// TIA Portal project "Projet3rob" (V15)

(* hardware
DEVICE "Station S7-1200_1"  S7-1200 Station
   slot 0: "Châssis_0"  S7-1200 Rack  Rack  V1.0
   slot 1: "PLC_1"  CPU 1212C DC/DC/DC  6ES7 212-1AE40-0XB0  V4.2
   slot 2: "DI 16/DQ 16x24VDC_1"  6ES7 223-1BL32-0XB0  V2.0
DEVICE "PC-System_1"  SIMATIC PC station
   slot 0: "Station PC SIMATIC"  Rail  SIMATIC PC-Station  V1.0
      slot 125: "Stationmanager"  Station_Manager  V6.0.4
   slot 1: "HMI_RT_1"  WinCC RT Advanced  6AV2 104-0xxxx-xxxx  15.0.0.0
      slot 33792: "Interface hôte"  Host interface
   slot 2: "IE Général_1"  IE General  IE_CP  V8.2.0
*)

// ===== PLC "PLC_1"  CPU 1212C DC/DC/DC =====

VAR_GLOBAL   // PLC tag table "Table de variables standard"
   "System_Byte" AT %MB1 : Byte;
   "FirstScan" AT %M1.0 : Bool;
   "DiagStatusUpdate" AT %M1.1 : Bool;
   "AlwaysTRUE" AT %M1.2 : Bool;
   "AlwaysFALSE" AT %M1.3 : Bool;
   "Clock_Byte" AT %MB0 : Byte;
   "Clock_10Hz" AT %M0.0 : Bool;
   "Clock_5Hz" AT %M0.1 : Bool;
   "Clock_2.5Hz" AT %M0.2 : Bool;
   "Clock_2Hz" AT %M0.3 : Bool;
   "Clock_1.25Hz" AT %M0.4 : Bool;
   "Clock_1Hz" AT %M0.5 : Bool;
   "Clock_0.625Hz" AT %M0.6 : Bool;
   "Clock_0.5Hz" AT %M0.7 : Bool;
   "Q_AUTO_ROBOT_DO_KEP" AT %M22.0 : Bool;
   "ACT_PRODUCT_DO" AT %MW210 : Word;
   "I_ROBOT_DO_KEP" AT %I3.0 : Bool;
   "M_ROBOT_DO_KEP" AT %M13.2 : Bool;
   "Q_MUNU_ROB_DO_KEP" AT %M22.2 : Bool;
END_VAR

VAR_GLOBAL   // PLC tag table "Input"
   "I_Mode" AT %I0.0 : Bool;
   "I_Run" AT %I0.1 : Bool;
   "I_Stop" AT %I0.2 : Bool;
   "I_CB_Vao" AT %I0.3 : Bool;
   "I_CB_Do" AT %I0.4 : Bool;
   "I_CB_Xanh" AT %I0.5 : Bool;
   "I_CB_Do1" AT %I0.6 : Bool;
   "I_CB_Xanh2" AT %I0.7 : Bool;
   "I_CB_Robot_Do_Phai" AT %I1.0 : Bool;
   "I_CB_Robot_Do_Trai" AT %I1.1 : Bool;
   "I_CB_Robot_Do_Giua" AT %I1.2 : Bool;
   "I_CB_Robot_Xanh_Phai" AT %I1.3 : Bool;
   "I_CB_Robot_Xanh_Trai" AT %I1.4 : Bool;
   "I_CB_Robot_Xanh_Giua" AT %I1.5 : Bool;
   "I_BT1" AT %I1.6 : Bool;
   "I_BT2" AT %I1.7 : Bool;
   "I_Xylanh_Do" AT %I2.0 : Bool;
   "I_Xylanh_Xanh" AT %I2.1 : Bool;
   "I_Robot_Do_Trai" AT %I2.2 : Bool;
   "I_Robot_Do_Phai" AT %I2.3 : Bool;
   "I_Robot_Do_Glua" AT %I2.4 : Bool;
   "I_Robot_Xanh_Trai" AT %I2.5 : Bool;
   "I_Robot_Xanh_Phai" AT %I2.6 : Bool;
   "I_Robot_Xanh_Glua" AT %I2.7 : Bool;
END_VAR

VAR_GLOBAL   // PLC tag table "M"
   "M_Mode" AT %M10.0 : Bool;
   "M_Run" AT %M10.1 : Bool;
   "M_Stop" AT %M10.2 : Bool;
   "M_CB_Vao" AT %M10.3 : Bool;
   "M_CB_Do" AT %M10.4 : Bool;
   "M_CB_Xanh" AT %M10.5 : Bool;
   "M_CB_Do1" AT %M10.6 : Bool;
   "M_CB_Xanh2" AT %M10.7 : Bool;
   "M_CB_Robot_Do_Phai" AT %M11.0 : Bool;
   "M_CB_Robot_Do_Trai" AT %M11.1 : Bool;
   "M_CB_Robot_Do_Giua" AT %M11.2 : Bool;
   "M_CB_Robot_Xanh_Phai" AT %M11.3 : Bool;
   "M_CB_Robot_Xanh_Trai" AT %M11.4 : Bool;
   "M_CB_Robot_Xanh_Giua" AT %M11.5 : Bool;
   "M_BT1" AT %M11.6 : Bool;
   "M_BT2" AT %M11.7 : Bool;
   "M_Xylanh_Do" AT %M12.0 : Bool;
   "M_Xylanh_Xanh" AT %M12.1 : Bool;
   "M_Robot_Do_Trai" AT %M12.2 : Bool;
   "M_Robot_Do_Phai" AT %M12.3 : Bool;
   "M_Robot_Do_Glua" AT %M12.4 : Bool;
   "M_Robot_Xanh_Trai" AT %M12.5 : Bool;
   "M_Robot_Xanh_Phai" AT %M12.6 : Bool;
   "M_Robot_Xanh_Glua" AT %M12.7 : Bool;
   "M_Simulation" AT %M13.0 : Bool;
   "M_Reset" AT %M13.1 : Bool;
END_VAR

VAR_GLOBAL   // PLC tag table "OUTPUT"
   "Q_Lamp_Auto" AT %Q0.0 : Bool;
   "Q_Lamp_Manu" AT %Q0.1 : Bool;
   "Q_Lamp_Running" AT %Q0.2 : Bool;
   "Q_Lamp_Stop" AT %Q0.3 : Bool;
   "Q_BT1" AT %Q0.4 : Bool;
   "Q_BT2" AT %Q0.5 : Bool;
   "Q_Xylanh_Do" AT %Q0.6 : Bool;
   "Q_Xylanh_Xanh" AT %Q0.7 : Bool;
   "Q_Robot_Do_Trai" AT %Q1.0 : Bool;
   "Q_Robot_Do_Phai" AT %Q1.1 : Bool;
   "Q_Robot_Xanh_Trai" AT %Q1.2 : Bool;
   "Q_Robot_Xanh_Phai" AT %Q1.3 : Bool;
END_VAR

VAR_GLOBAL   // PLC tag table "Xlanh P"
   "P1" AT %M40.0 : Bool;
   "P2" AT %M40.1 : Bool;
   "P3" AT %M40.2 : Bool;
   "P4" AT %M40.3 : Bool;
   "P5" AT %M40.4 : Bool;
   "P6" AT %M40.5 : Bool;
   "P7" AT %M40.6 : Bool;
   "P8" AT %M40.7 : Bool;
   "P9" AT %M41.0 : Bool;
   "P10" AT %M41.1 : Bool;
   "P11" AT %M41.2 : Bool;
   "P12" AT %M41.3 : Bool;
   "P13" AT %M41.4 : Bool;
   "P14" AT %M41.5 : Bool;
   "P15" AT %M41.6 : Bool;
   "P16" AT %M41.7 : Bool;
   "P17" AT %M42.0 : Bool;
   "P18" AT %M42.1 : Bool;
   "P19" AT %M42.2 : Bool;
   "P20" AT %M42.3 : Bool;
   "P21" AT %M42.4 : Bool;
   "P22" AT %M42.5 : Bool;
   "P23" AT %M42.6 : Bool;
   "P24" AT %M42.7 : Bool;
   "P25" AT %M43.0 : Bool;
   "P26" AT %M43.1 : Bool;
   "P27" AT %M43.2 : Bool;
   "P28" AT %M43.3 : Bool;
   "P29" AT %M43.4 : Bool;
   "P30" AT %M43.5 : Bool;
END_VAR

VAR_GLOBAL   // PLC tag table "TRING GIAN"
   "Q_Auto_BT1" AT %M20.0 : Bool;
   "Q_Auto_BT2" AT %M20.1 : Bool;
   "Q_Auto_Xylanh_Do" AT %M20.2 : Bool;
   "Q_Auto_Xylanh_Xanh" AT %M20.3 : Bool;
   "Q_Auto_Robot_Do_Trai" AT %M20.4 : Bool;
   "Q_Auto_Robot_Do_Phai" AT %M20.5 : Bool;
   "Q_Auto_Robot_Xanh_Trai" AT %M20.6 : Bool;
   "Q_Auto_Robot_Xanh_Phai" AT %M20.7 : Bool;
   "Q_Manu_BT1" AT %M21.0 : Bool;
   "Q_Manu_BT2" AT %M21.1 : Bool;
   "Q_Manu_Xylanh_Do" AT %M21.2 : Bool;
   "Q_Manu_Xylanh_Xanh" AT %M21.3 : Bool;
   "Q_Manu_Robot_Do_Trai" AT %M21.4 : Bool;
   "Q_Manu_Robot_Do_Phai" AT %M21.5 : Bool;
   "Q_Manu_Robot_Xanh_Trai" AT %M21.6 : Bool;
   "Q_Manu_Robot_Xanh_Phai" AT %M21.7 : Bool;
END_VAR

VAR_GLOBAL   // PLC tag table "DU MUE"
   "Act_Count_Vao" AT %MW200 : Int;
   "Act_Count_Do" AT %MW202 : Int;
   "Act_Count_Do1" AT %MW204 : Int;
   "Act_Count_Xnah" AT %MW206 : Int;
   "Act_Count_Xnah1" AT %MW208 : Int;
END_VAR

VAR_GLOBAL   // PLC tag table "Table de variables_1"
   "ROBOT_DO_AUTO_STEP1" AT %M25.0 : Bool;
   "ROBOT_DO_AUTO_STEP2" AT %M25.1 : Bool;
   "ROBOT_DO_AUTO_STEP3" AT %M25.2 : Bool;
   "ROBOT_DO_AUTO_STEP4" AT %M25.3 : Bool;
   "ROBOT_DO_AUTO_STEP5" AT %M25.4 : Bool;
   "ROBOT_XNAH_AUTO_STEP1" AT %M25.5 : Bool;
   "ROBOT_XNAH_AUTO_STEP2" AT %M25.6 : Bool;
   "ROBOT_XNAH_AUTO_STEP3" AT %M25.7 : Bool;
   "ROBOT_XNAH_AUTO_STEP4" AT %M26.0 : Bool;
   "ROBOT_XNAH_AUTO_STEP5" AT %M26.1 : Bool;
END_VAR

// folder: System blocks/Program resources

DATA_BLOCK "IEC_Timer_0_DB"   // DB1
{ S7_Optimized_Access := 'TRUE' }
AUTHOR : Simatic
FAMILY : IEC
NAME : IEC_TMR
VERSION : 1.0
// stored: InstanceOfName IEC_TIMER
"IEC_TIMER"
BEGIN
END_DATA_BLOCK

DATA_BLOCK "TIMER_DELYE_SET_XL_DO"   // DB2
{ S7_Optimized_Access := 'TRUE' }
AUTHOR : Simatic
FAMILY : IEC
NAME : IEC_TMR
VERSION : 1.0
// stored: InstanceOfName IEC_TIMER
"IEC_TIMER"
BEGIN
END_DATA_BLOCK

DATA_BLOCK "TIMER_XL_DO"   // DB3
{ S7_Optimized_Access := 'TRUE' }
AUTHOR : Simatic
FAMILY : IEC
NAME : IEC_TMR
VERSION : 1.0
// stored: InstanceOfName IEC_TIMER
"IEC_TIMER"
BEGIN
END_DATA_BLOCK

DATA_BLOCK "TIME_KEP_DO1"   // DB4
{ S7_Optimized_Access := 'TRUE' }
AUTHOR : Simatic
FAMILY : IEC
NAME : IEC_TMR
VERSION : 1.0
// stored: InstanceOfName IEC_TIMER
"IEC_TIMER"
BEGIN
END_DATA_BLOCK

DATA_BLOCK "TIMER_KEP_DO2"   // DB5
{ S7_Optimized_Access := 'TRUE' }
AUTHOR : Simatic
FAMILY : IEC
NAME : IEC_TMR
VERSION : 1.0
// stored: InstanceOfName IEC_TIMER
"IEC_TIMER"
BEGIN
END_DATA_BLOCK

DATA_BLOCK "IEC_Timer_0_DB_1"   // DB6
{ S7_Optimized_Access := 'TRUE' }
AUTHOR : Simatic
FAMILY : IEC
NAME : IEC_TMR
VERSION : 1.0
// stored: InstanceOfName IEC_TIMER
"IEC_TIMER"
BEGIN
END_DATA_BLOCK

DATA_BLOCK "TIMER_DELYE_SET_XL_XNAH"   // DB7
{ S7_Optimized_Access := 'TRUE' }
AUTHOR : Simatic
FAMILY : IEC
NAME : IEC_TMR
VERSION : 1.0
// stored: InstanceOfName IEC_TIMER
"IEC_TIMER"
BEGIN
END_DATA_BLOCK

DATA_BLOCK "TIMER_XL_XANH"   // DB8
{ S7_Optimized_Access := 'TRUE' }
AUTHOR : Simatic
FAMILY : IEC
NAME : IEC_TMR
VERSION : 1.0
// stored: InstanceOfName IEC_TIMER
"IEC_TIMER"
BEGIN
END_DATA_BLOCK

// folder: (top level)

FUNCTION "FC_Auto" : Void   // FC1, LAD
{ S7_Optimized_Access := 'TRUE' }
VERSION : 0.1
   VAR_TEMP   // added for the SCL form of the ladder/FBD networks
      _w1 : Bool;
      _w2 : Bool;
      _w3 : Bool;
      _w4 : Bool;
      _w5 : Bool;
      _w6 : Bool;
      _w7 : Bool;
      _w8 : Bool;
      _w9 : Bool;
      _w10 : Bool;
      _w11 : Bool;
      _w12 : Bool;
      _w13 : Bool;
      _w14 : Bool;
   END_VAR
BEGIN

REGION Network 1
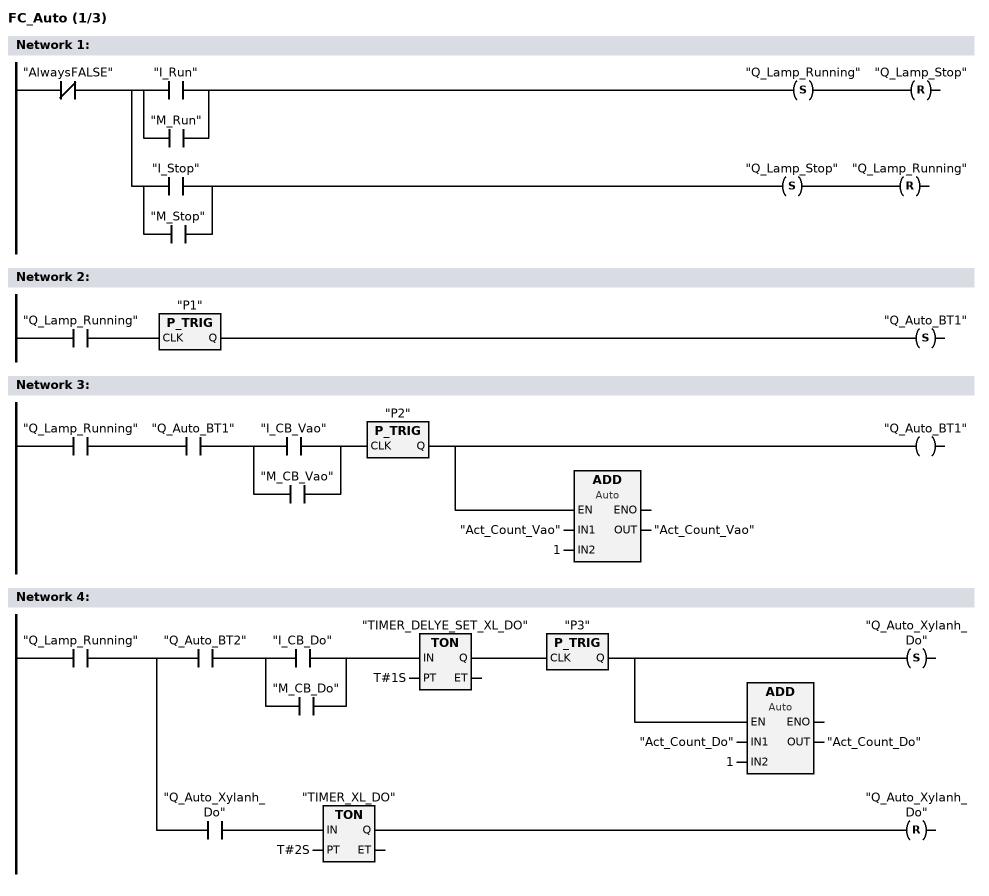
   RUNG wire#powerrail
      I_Contact( "AlwaysFALSE" )
      wire#w1
      Contact( "I_Run" )
      wire#w2
      S_Coil( "Q_Lamp_Running" )
      R_Coil( "Q_Lamp_Stop" )
   END_RUNG
   RUNG wire#w1
      Contact( "M_Run" )
   END_RUNG wire#w2
   RUNG wire#w1
      Contact( "I_Stop" )
      wire#w3
      S_Coil( "Q_Lamp_Stop" )
      R_Coil( "Q_Lamp_Running" )
   END_RUNG
   RUNG wire#w1
      Contact( "M_Stop" )
   END_RUNG wire#w3
   // the same network as SCL:
   IF NOT "AlwaysFALSE" AND ("I_Run" OR "M_Run") THEN
       "Q_Lamp_Running" := TRUE;
       "Q_Lamp_Stop" := FALSE;
   END_IF;
   IF NOT "AlwaysFALSE" AND ("I_Stop" OR "M_Stop") THEN
       "Q_Lamp_Stop" := TRUE;
       "Q_Lamp_Running" := FALSE;
   END_IF;
END_REGION

REGION Network 2
   RUNG wire#powerrail
      Contact( "Q_Lamp_Running" )
      P_Trig( "P1" )
      S_Coil( "Q_Auto_BT1" )
   END_RUNG
   // the same network as SCL:
   #_w1 := "Q_Lamp_Running" AND NOT "P1";   // rising edge
   "P1" := "Q_Lamp_Running";
   IF #_w1 THEN "Q_Auto_BT1" := TRUE; END_IF;
END_REGION

REGION Network 3
   RUNG wire#powerrail
      Contact( "Q_Lamp_Running" )
      Contact( "Q_Auto_BT1" )
      wire#w1
      Contact( "I_CB_Vao" )
      wire#w2
      P_Trig( "P2" )
      wire#w3
      Coil( "Q_Auto_BT1" )
   END_RUNG
   RUNG wire#w1
      Contact( "M_CB_Vao" )
   END_RUNG wire#w2
   RUNG wire#w3
      Add(in1 := "Act_Count_Vao", in2 := 1, out => "Act_Count_Vao")
   END_RUNG
   // the same network as SCL:
   #_w1 := "Q_Lamp_Running" AND "Q_Auto_BT1" AND ("I_CB_Vao" OR "M_CB_Vao");
   #_w2 := #_w1 AND NOT "P2";   // rising edge
   "P2" := #_w1;
   "Q_Auto_BT1" := #_w2;
   IF #_w2 THEN "Act_Count_Vao" := "Act_Count_Vao" + 1; END_IF;
END_REGION

REGION Network 4
   "TIMER_DELYE_SET_XL_DO".TON(IN := "Q_Lamp_Running" AND "Q_Auto_BT2" AND ("I_CB_Do" OR "M_CB_Do"), PT := T#1S);
   #_w1 := "TIMER_DELYE_SET_XL_DO".Q AND NOT "P3";   // rising edge
   "P3" := "TIMER_DELYE_SET_XL_DO".Q;
   IF #_w1 THEN
       "Q_Auto_Xylanh_Do" := TRUE;
       "Act_Count_Do" := "Act_Count_Do" + 1;
   END_IF;
   "TIMER_XL_DO".TON(IN := "Q_Lamp_Running" AND "Q_Auto_Xylanh_Do", PT := T#2S);
   IF "TIMER_XL_DO".Q THEN "Q_Auto_Xylanh_Do" := FALSE; END_IF;
END_REGION

REGION Network 5
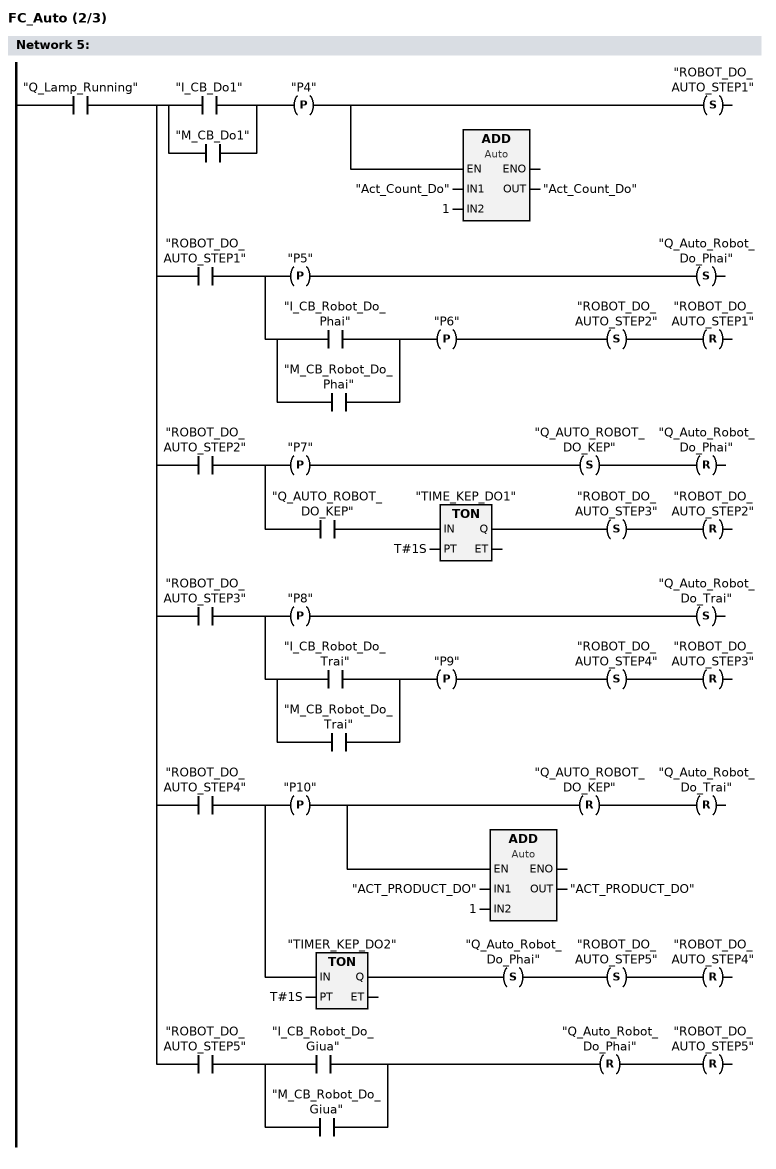
   #_w1 := "Q_Lamp_Running" AND ("I_CB_Do1" OR "M_CB_Do1");
   #_w2 := #_w1 AND NOT "P4";   // rising edge
   "P4" := #_w1;
   IF #_w2 THEN
       "ROBOT_DO_AUTO_STEP1" := TRUE;
       "Act_Count_Do" := "Act_Count_Do" + 1;
   END_IF;
   #_w3 := "Q_Lamp_Running" AND "ROBOT_DO_AUTO_STEP1";
   #_w4 := #_w3 AND NOT "P5";   // rising edge
   "P5" := #_w3;
   IF #_w4 THEN "Q_Auto_Robot_Do_Phai" := TRUE; END_IF;
   #_w5 := #_w3 AND ("I_CB_Robot_Do_Phai" OR "M_CB_Robot_Do_Phai");
   #_w6 := #_w5 AND NOT "P6";   // rising edge
   "P6" := #_w5;
   IF #_w6 THEN
       "ROBOT_DO_AUTO_STEP2" := TRUE;
       "ROBOT_DO_AUTO_STEP1" := FALSE;
   END_IF;
   #_w7 := "Q_Lamp_Running" AND "ROBOT_DO_AUTO_STEP2";
   #_w8 := #_w7 AND NOT "P7";   // rising edge
   "P7" := #_w7;
   IF #_w8 THEN
       "Q_AUTO_ROBOT_DO_KEP" := TRUE;
       "Q_Auto_Robot_Do_Phai" := FALSE;
   END_IF;
   "TIME_KEP_DO1".TON(IN := #_w7 AND "Q_AUTO_ROBOT_DO_KEP", PT := T#1S);
   IF "TIME_KEP_DO1".Q THEN
       "ROBOT_DO_AUTO_STEP3" := TRUE;
       "ROBOT_DO_AUTO_STEP2" := FALSE;
   END_IF;
   #_w9 := "Q_Lamp_Running" AND "ROBOT_DO_AUTO_STEP3";
   #_w10 := #_w9 AND NOT "P8";   // rising edge
   "P8" := #_w9;
   IF #_w10 THEN "Q_Auto_Robot_Do_Trai" := TRUE; END_IF;
   #_w11 := #_w9 AND ("I_CB_Robot_Do_Trai" OR "M_CB_Robot_Do_Trai");
   #_w12 := #_w11 AND NOT "P9";   // rising edge
   "P9" := #_w11;
   IF #_w12 THEN
       "ROBOT_DO_AUTO_STEP4" := TRUE;
       "ROBOT_DO_AUTO_STEP3" := FALSE;
   END_IF;
   #_w13 := "Q_Lamp_Running" AND "ROBOT_DO_AUTO_STEP4";
   #_w14 := #_w13 AND NOT "P10";   // rising edge
   "P10" := #_w13;
   IF #_w14 THEN
       "Q_AUTO_ROBOT_DO_KEP" := FALSE;
       "Q_Auto_Robot_Do_Trai" := FALSE;
       "ACT_PRODUCT_DO" := "ACT_PRODUCT_DO" + 1;
   END_IF;
   "TIMER_KEP_DO2".TON(IN := #_w13, PT := T#1S);
   IF "TIMER_KEP_DO2".Q THEN
       "Q_Auto_Robot_Do_Phai" := TRUE;
       "ROBOT_DO_AUTO_STEP5" := TRUE;
       "ROBOT_DO_AUTO_STEP4" := FALSE;
   END_IF;
   IF "Q_Lamp_Running" AND "ROBOT_DO_AUTO_STEP5" AND ("I_CB_Robot_Do_Giua" OR "M_CB_Robot_Do_Giua") THEN
       "Q_Auto_Robot_Do_Phai" := FALSE;
       "ROBOT_DO_AUTO_STEP5" := FALSE;
   END_IF;
END_REGION

REGION Network 6
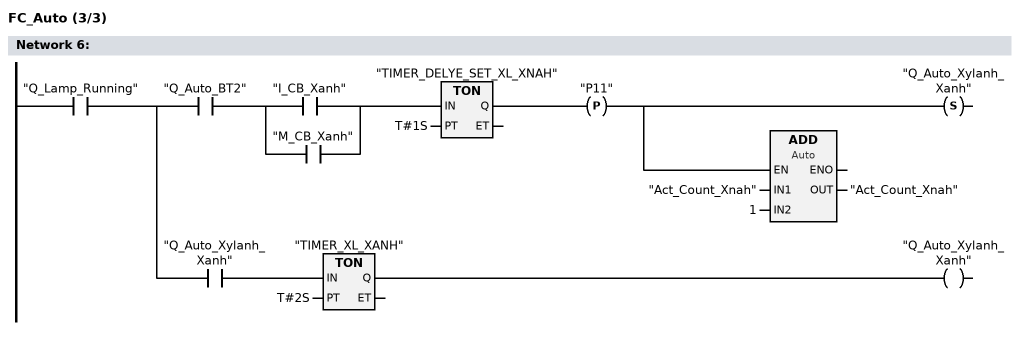
   "TIMER_DELYE_SET_XL_XNAH".TON(IN := "Q_Lamp_Running" AND "Q_Auto_BT2" AND ("I_CB_Xanh" OR "M_CB_Xanh"),
                           PT := T#1S);
   #_w1 := "TIMER_DELYE_SET_XL_XNAH".Q AND NOT "P11";   // rising edge
   "P11" := "TIMER_DELYE_SET_XL_XNAH".Q;
   IF #_w1 THEN
       "Q_Auto_Xylanh_Xanh" := TRUE;
       "Act_Count_Xnah" := "Act_Count_Xnah" + 1;
   END_IF;
   "TIMER_XL_XANH".TON(IN := "Q_Lamp_Running" AND "Q_Auto_Xylanh_Xanh", PT := T#2S);
   "Q_Auto_Xylanh_Xanh" := "TIMER_XL_XANH".Q;
END_REGION
END_FUNCTION

FUNCTION "FC_Manu" : Void   // FC2, LAD
{ S7_Optimized_Access := 'TRUE' }
VERSION : 0.1
   VAR_TEMP   // added for the SCL form of the ladder/FBD networks
      _w1 : Bool;
      _w2 : Bool;
      _w3 : Bool;
      _w4 : Bool;
   END_VAR
BEGIN

REGION Network 1
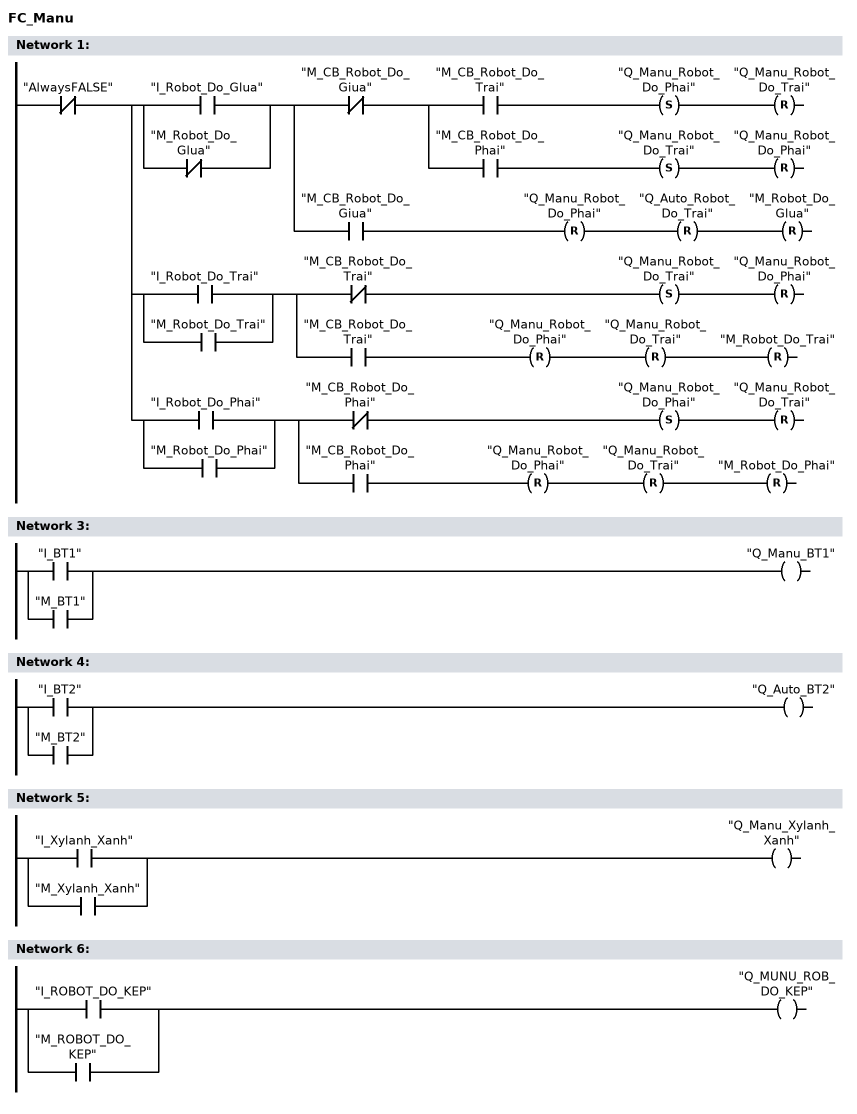
   RUNG wire#powerrail
      I_Contact( "AlwaysFALSE" )
      wire#w1
      Contact( "I_Robot_Do_Glua" )
      wire#w2
      I_Contact( "M_CB_Robot_Do_Giua" )
      wire#w3
      Contact( "M_CB_Robot_Do_Trai" )
      S_Coil( "Q_Manu_Robot_Do_Phai" )
      R_Coil( "Q_Manu_Robot_Do_Trai" )
   END_RUNG
   RUNG wire#w1
      I_Contact( "M_Robot_Do_Glua" )
   END_RUNG wire#w2
   RUNG wire#w3
      Contact( "M_CB_Robot_Do_Phai" )
      S_Coil( "Q_Manu_Robot_Do_Trai" )
      R_Coil( "Q_Manu_Robot_Do_Phai" )
   END_RUNG
   RUNG wire#w2
      Contact( "M_CB_Robot_Do_Giua" )
      R_Coil( "Q_Manu_Robot_Do_Phai" )
      R_Coil( "Q_Auto_Robot_Do_Trai" )
      R_Coil( "M_Robot_Do_Glua" )
   END_RUNG
   RUNG wire#w1
      Contact( "I_Robot_Do_Trai" )
      wire#w4
      I_Contact( "M_CB_Robot_Do_Trai" )
      S_Coil( "Q_Manu_Robot_Do_Trai" )
      R_Coil( "Q_Manu_Robot_Do_Phai" )
   END_RUNG
   RUNG wire#w1
      Contact( "M_Robot_Do_Trai" )
   END_RUNG wire#w4
   RUNG wire#w4
      Contact( "M_CB_Robot_Do_Trai" )
      R_Coil( "Q_Manu_Robot_Do_Phai" )
      R_Coil( "Q_Manu_Robot_Do_Trai" )
      R_Coil( "M_Robot_Do_Trai" )
   END_RUNG
   RUNG wire#w1
      Contact( "I_Robot_Do_Phai" )
      wire#w5
      I_Contact( "M_CB_Robot_Do_Phai" )
      S_Coil( "Q_Manu_Robot_Do_Phai" )
      R_Coil( "Q_Manu_Robot_Do_Trai" )
   END_RUNG
   RUNG wire#w1
      Contact( "M_Robot_Do_Phai" )
   END_RUNG wire#w5
   RUNG wire#w5
      Contact( "M_CB_Robot_Do_Phai" )
      R_Coil( "Q_Manu_Robot_Do_Phai" )
      R_Coil( "Q_Manu_Robot_Do_Trai" )
      R_Coil( "M_Robot_Do_Phai" )
   END_RUNG
   // the same network as SCL:
   #_w1 := NOT "AlwaysFALSE" AND ("I_Robot_Do_Glua" OR NOT "M_Robot_Do_Glua");
   #_w2 := #_w1 AND NOT "M_CB_Robot_Do_Giua";
   IF #_w2 AND "M_CB_Robot_Do_Trai" THEN
       "Q_Manu_Robot_Do_Phai" := TRUE;
       "Q_Manu_Robot_Do_Trai" := FALSE;
   END_IF;
   IF #_w2 AND "M_CB_Robot_Do_Phai" THEN
       "Q_Manu_Robot_Do_Trai" := TRUE;
       "Q_Manu_Robot_Do_Phai" := FALSE;
   END_IF;
   IF #_w1 AND "M_CB_Robot_Do_Giua" THEN
       "Q_Manu_Robot_Do_Phai" := FALSE;
       "Q_Auto_Robot_Do_Trai" := FALSE;
       "M_Robot_Do_Glua" := FALSE;
   END_IF;
   #_w3 := NOT "AlwaysFALSE" AND ("I_Robot_Do_Trai" OR "M_Robot_Do_Trai");
   IF #_w3 AND NOT "M_CB_Robot_Do_Trai" THEN
       "Q_Manu_Robot_Do_Trai" := TRUE;
       "Q_Manu_Robot_Do_Phai" := FALSE;
   END_IF;
   IF #_w3 AND "M_CB_Robot_Do_Trai" THEN
       "Q_Manu_Robot_Do_Phai" := FALSE;
       "Q_Manu_Robot_Do_Trai" := FALSE;
       "M_Robot_Do_Trai" := FALSE;
   END_IF;
   #_w4 := NOT "AlwaysFALSE" AND ("I_Robot_Do_Phai" OR "M_Robot_Do_Phai");
   IF #_w4 AND NOT "M_CB_Robot_Do_Phai" THEN
       "Q_Manu_Robot_Do_Phai" := TRUE;
       "Q_Manu_Robot_Do_Trai" := FALSE;
   END_IF;
   IF #_w4 AND "M_CB_Robot_Do_Phai" THEN
       "Q_Manu_Robot_Do_Phai" := FALSE;
       "Q_Manu_Robot_Do_Trai" := FALSE;
       "M_Robot_Do_Phai" := FALSE;
   END_IF;
END_REGION

REGION Network 3
   RUNG wire#powerrail
      Contact( "I_BT1" )
      wire#w1
      Coil( "Q_Manu_BT1" )
   END_RUNG
   RUNG wire#powerrail
      Contact( "M_BT1" )
   END_RUNG wire#w1
   // the same network as SCL:
   "Q_Manu_BT1" := "I_BT1" OR "M_BT1";
END_REGION

REGION Network 4
   RUNG wire#powerrail
      Contact( "I_BT2" )
      wire#w1
      Coil( "Q_Auto_BT2" )
   END_RUNG
   RUNG wire#powerrail
      Contact( "M_BT2" )
   END_RUNG wire#w1
   // the same network as SCL:
   "Q_Auto_BT2" := "I_BT2" OR "M_BT2";
END_REGION

REGION Network 5
   RUNG wire#powerrail
      Contact( "I_Xylanh_Xanh" )
      wire#w1
      Coil( "Q_Manu_Xylanh_Xanh" )
   END_RUNG
   RUNG wire#powerrail
      Contact( "M_Xylanh_Xanh" )
   END_RUNG wire#w1
   // the same network as SCL:
   "Q_Manu_Xylanh_Xanh" := "I_Xylanh_Xanh" OR "M_Xylanh_Xanh";
END_REGION

REGION Network 6
   RUNG wire#powerrail
      Contact( "I_ROBOT_DO_KEP" )
      wire#w1
      Coil( "Q_MUNU_ROB_DO_KEP" )
   END_RUNG
   RUNG wire#powerrail
      Contact( "M_ROBOT_DO_KEP" )
   END_RUNG wire#w1
   // the same network as SCL:
   "Q_MUNU_ROB_DO_KEP" := "I_ROBOT_DO_KEP" OR "M_ROBOT_DO_KEP";
END_REGION
END_FUNCTION

FUNCTION "FC_SIMULATION" : Void   // FC3, LAD
{ S7_Optimized_Access := 'TRUE' }
VERSION : 0.1
BEGIN
END_FUNCTION

FUNCTION "FC_OUTPUT" : Void   // FC4, LAD
{ S7_Optimized_Access := 'TRUE' }
VERSION : 0.1
BEGIN
END_FUNCTION

ORGANIZATION_BLOCK "Main"   // OB1, LAD, ProgramCycle
TITLE = "Main Program Sweep (Cycle)"
{ S7_Optimized_Access := 'TRUE' }
VERSION : 0.1
   VAR_INPUT
      Initial_Call : Bool;   // Initial call of this OB
      Remanence : Bool;   // =True, if remanent data are available
   END_VAR
BEGIN

REGION Network 1
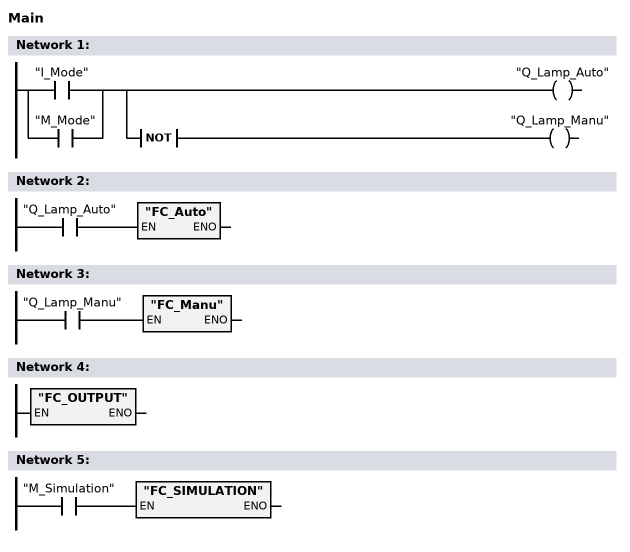
   RUNG wire#powerrail
      Contact( "I_Mode" )
      wire#w1
      Coil( "Q_Lamp_Auto" )
   END_RUNG
   RUNG wire#powerrail
      Contact( "M_Mode" )
   END_RUNG wire#w1
   RUNG wire#w1
      Not()
      Coil( "Q_Lamp_Manu" )
   END_RUNG
   // the same network as SCL:
   "Q_Lamp_Auto" := "I_Mode" OR "M_Mode";
   "Q_Lamp_Manu" := NOT "Q_Lamp_Auto";
END_REGION

REGION Network 2
   RUNG wire#powerrail
      Contact( "Q_Lamp_Auto" )
      "FC_Auto"()
   END_RUNG
   // the same network as SCL:
   IF "Q_Lamp_Auto" THEN "FC_Auto"(); END_IF;
END_REGION

REGION Network 3
   RUNG wire#powerrail
      Contact( "Q_Lamp_Manu" )
      "FC_Manu"()
   END_RUNG
   // the same network as SCL:
   IF "Q_Lamp_Manu" THEN "FC_Manu"(); END_IF;
END_REGION

REGION Network 4
   RUNG wire#powerrail
      "FC_OUTPUT"()
   END_RUNG
   // the same network as SCL:
   "FC_OUTPUT"();
END_REGION

REGION Network 5
   RUNG wire#powerrail
      Contact( "M_Simulation" )
      "FC_SIMULATION"()
   END_RUNG
   // the same network as SCL:
   IF "M_Simulation" THEN "FC_SIMULATION"(); END_IF;
END_REGION
END_ORGANIZATION_BLOCK

ORGANIZATION_BLOCK "Startup"   // OB100, LAD, Startup
TITLE = "Complete Restart"
{ S7_Optimized_Access := 'TRUE' }
VERSION : 0.1
   VAR_INPUT
      LostRetentive : Bool;   // True if retentive data are lost
      LostRTC : Bool;   // True if date and time are lost
   END_VAR
BEGIN
END_ORGANIZATION_BLOCK

(* ===== HMI "HMI_RT_1" =====
system functions are stored by id; their names below are inferred from use
connection "HMI_Liaison_1": ETHERNET, S7_1200_OMS

HMI tags "Table de variables standard"
   "Q_BT2" : Bool = PLC Q_BT2 AT %Q0.5, 1 s
   "Q_BT1" : Bool = PLC Q_BT1 AT %Q0.4, 1 s
   "M_CB_Vao" : Bool = PLC M_CB_Vao AT %M10.3, 1 s
   "M_CB_Do" : Bool = PLC M_CB_Do AT %M10.4, 1 s
   "M_CB_Xanh" : Bool = PLC M_CB_Xanh AT %M10.5, 1 s
   "M_CB_Do1" : Bool = PLC M_CB_Do1 AT %M10.6, 1 s
   "M_CB_Xanh1" : Bool = PLC M_CB_Xanh2 AT %M10.7, 1 s
   "M_CB_Robot_Do_Trai" : Bool = PLC M_CB_Robot_Do_Trai AT %M11.1, 1 s
   "M_CB_Robot_Do_Giua" : Bool = PLC M_CB_Robot_Do_Giua AT %M11.2, 1 s
   "M_CB_Robot_Do_Phai" : Bool = PLC M_CB_Robot_Do_Phai AT %M11.0, 1 s
   "M_CB_Robot_Xanh_Trai" : Bool = PLC M_CB_Robot_Xanh_Trai AT %M11.4, 1 s
   "M_CB_Robot_Xanh_Giua" : Bool = PLC M_CB_Robot_Xanh_Giua AT %M11.5, 1 s
   "M_CB_Robot_Xanh_Phai" : Bool = PLC M_CB_Robot_Xanh_Phai AT %M11.3, 1 s
   "Q_Xylanh_Do" : Bool = PLC Q_Xylanh_Do AT %Q0.6, 1 s
   "Q_Xylanh_Xanh" : Bool = PLC Q_Xylanh_Xanh AT %Q0.7, 1 s
   "M_Simulation" : Bool = PLC M_Simulation AT %M13.0, 1 s
   "M_Mode" : Bool = PLC M_Mode AT %M10.0, 1 s
   "M_Run" : Bool = PLC M_Run AT %M10.1, 1 s
   "M_Stop" : Bool = PLC M_Stop AT %M10.2, 1 s
   "M_Reset" : Bool = PLC M_Reset AT %M13.1, 1 s
   "Q_Lamp_Auto" : Bool = PLC Q_Lamp_Auto AT %Q0.0, 1 s
   "Q_Lamp_Manu" : Bool = PLC Q_Lamp_Manu AT %Q0.1, 1 s
   "Q_Lamp_Running" : Bool = PLC Q_Lamp_Running AT %Q0.2, 1 s
   "Q_Lamp_Stop" : Bool = PLC Q_Lamp_Stop AT %Q0.3, 1 s
   "M_BT1" : Bool = PLC M_BT1 AT %M11.6, 1 s
   "M_BT2" : Bool = PLC M_BT2 AT %M11.7, 1 s
   "M_Xylanh_Do" : Bool = PLC M_Xylanh_Do AT %M12.0, 1 s
   "M_Xylanh_Xanh" : Bool = PLC M_Xylanh_Xanh AT %M12.1, 1 s
   "M_Robot_Do_Phai" : Bool = PLC M_Robot_Do_Phai AT %M12.3, 1 s
   "M_Robot_Do_Glua" : Bool = PLC M_Robot_Do_Glua AT %M12.4, 1 s
   "M_Robot_Do_Trai" : Bool = PLC M_Robot_Do_Trai AT %M12.2, 1 s
   "M_Robot_Xanh_Phai" : Bool = PLC M_Robot_Xanh_Phai AT %M12.6, 1 s
   "M_Robot_Xanh_Glua" : Bool = PLC M_Robot_Xanh_Glua AT %M12.7, 1 s
   "M_Robot_Xanh_Trai" : Bool = PLC M_Robot_Xanh_Trai AT %M12.5, 1 s
   "Q_Robot_Xanh_Trai" : Bool = PLC Q_Robot_Xanh_Trai AT %Q1.2, 1 s
   "Q_Robot_Xanh_Phai" : Bool = PLC Q_Robot_Xanh_Phai AT %Q1.3, 1 s
   "Q_Robot_Do_Trai" : Bool = PLC Q_Robot_Do_Trai AT %Q1.0, 1 s
   "Q_Robot_Do_Phai" : Bool = PLC Q_Robot_Do_Phai AT %Q1.1, 1 s

screen "Vue_1" 1024x1280
   TextField "Champ de texte_1" at 370,18 size 186x22; Text 'TIA PORTAL + S7-1200'
   SymbolLibrary "Bibliothèque des icônes_2" at 257,256 size 212x54
      Appearance <- "Q_BT2"
   SymbolLibrary "Bibliothèque des icônes_3" at 436,255 size 215x54
      Appearance <- "Q_BT2"
   SymbolLibrary "Bibliothèque des icônes_4" at 21,251 size 263x54
      Appearance <- "Q_BT1"
   SymbolLibrary "Bibliothèque des icônes_5" at 172,181 size 27x47
      Appearance <- "M_CB_Vao"
   SymbolLibrary "Bibliothèque des icônes_6" at 37,308 size 57x60
      Appearance <- "Q_BT1"
   SymbolLibrary "Bibliothèque des icônes_8" at 358,176 size 27x57
      Appearance <- "M_CB_Do"
   Group "Group_2" at 434,141 size 78x66
   Polygon "Polygone_7" at 247,376 size 114x77
      Visibility <- "M_CB_Robot_Do_Phai"
   Polygon "Polygone_10" at 125,410 size 124x46
      Visibility <- "M_CB_Robot_Do_Trai"
   Rectangle "Rectangle_9" at 248,409 size 20x45
      Visibility <- "M_CB_Robot_Do_Giua"
   Circle "Cercle_2" at 333,420 size 10x10
      Appearance <- "M_CB_Robot_Do_Phai"
   Circle "Cercle_4" at 251,410 size 10x10
      Appearance <- "M_CB_Robot_Do_Giua"
   Circle "Cercle_5" at 151,428 size 10x10
      Appearance <- "M_CB_Robot_Do_Trai"
   SymbolLibrary "Bibliothèque des icônes_9" at 70,437 size 87x60
   SymbolLibrary "Bibliothèque des icônes_10" at 370,364 size 69x29
      Appearance <- "M_CB_Do1"
   IOField "Champ d'E/S_1" at 37,157 size 96x32; FormatPattern 9999999
   IOField "Champ d'E/S_2" at 330,141 size 96x32; FormatPattern 9999999
   IOField "Champ d'E/S_3" at 359,405 size 96x32; FormatPattern 9999999
   TextField "Champ de texte_2" at 133,156 size 39x22; Text '[SP]'
   TextField "Champ de texte_3" at 366,120 size 39x22; Text '[SP]'
   TextField "Champ de texte_4" at 383,440 size 39x22; Text '[SP]'
   SymbolLibrary "Bibliothèque des icônes_11" at 616,254 size 237x55
      Appearance <- "Q_BT2"
   SymbolLibrary "Bibliothèque des icônes_12" at 803,308 size 57x60
      Appearance <- "Q_BT2"
   SymbolLibrary "Bibliothèque des icônes_13" at 719,181 size 27x57
      Appearance <- "M_CB_Xanh"
   Group "Group_1" at 795,146 size 78x66
   Polygon "Polygone_18" at 629,382 size 94x80
      Visibility <- "M_CB_Robot_Xanh_Phai"
   Polygon "Polygone_19" at 486,402 size 140x55
      Visibility <- "M_CB_Robot_Xanh_Trai"
   Rectangle "Rectangle_15" at 609,414 size 20x45
      Visibility <- "M_CB_Robot_Xanh_Giua"
   Circle "Cercle_8" at 694,425 size 10x10
      Appearance <- "M_CB_Robot_Xanh_Phai"
   Circle "Cercle_9" at 612,415 size 10x10
      Appearance <- "M_CB_Robot_Xanh_Giua"
   Circle "Cercle_10" at 512,433 size 10x10
      Appearance <- "M_CB_Robot_Xanh_Trai"
   SymbolLibrary "Bibliothèque des icônes_14" at 436,468 size 87x60
   SymbolLibrary "Bibliothèque des icônes_15" at 734,368 size 69x29
      Appearance <- "M_CB_Xanh1"
   IOField "Champ d'E/S_4" at 691,146 size 96x32; FormatPattern 9999999
   IOField "Champ d'E/S_5" at 732,429 size 96x32; FormatPattern 9999999
   TextField "Champ de texte_5" at 727,125 size 39x22; Text '[SP]'
   TextField "Champ de texte_6" at 756,459 size 39x22; Text '[SP]'
   Group "Group" at 691,288 size 81x69
   IOField "Champ d'E/S_6" at 427,536 size 96x32; FormatPattern 9999999
   IOField "Champ d'E/S_7" at 53,508 size 96x32; FormatPattern 9999999
   TextField "Champ de texte_7" at 455,569 size 39x22; Text '[SP]'
   TextField "Champ de texte_8" at 81,545 size 39x22; Text '[SP]'
   Switch "Commutateur_1" at 711,596 size 118x63; CaptionText 'Switch'; TextOff 'MANU'; TextOn 'AUTO'
      on SwitchOff: SetBit("M_Mode")
      on SwitchOn: ResetBit("M_Mode")
      ProcessValue <- "M_Mode"
   Button "Bouton_1" at 721,682 size 96x32; TextOff 'RUN'
      on Press: SetBit("M_Run")
      on Release: ResetBit("M_Run")
   Button "Bouton_2" at 725,730 size 96x32; TextOff 'STOP'
      on Press: SetBit("M_Stop")
      on Release: ResetBit("M_Stop")
   Circle "Cercle_11" at 868,601 size 55x55
      Appearance <- "Q_Lamp_Auto"
   Circle "Cercle_12" at 929,599 size 57x57
      Appearance <- "Q_Lamp_Manu"
   Circle "Cercle_13" at 868,657 size 53x53
      Appearance <- "Q_Lamp_Running"
   Circle "Cercle_14" at 933,657 size 53x53
      Appearance <- "Q_Lamp_Running"
   TextField "Champ de texte_9" at 868,617 size 47x22; Text 'AUTO'
   TextField "Champ de texte_10" at 931,616 size 51x22; Text 'MANU'
   TextField "Champ de texte_11" at 876,670 size 39x22; Text 'RUN'
   TextField "Champ de texte_12" at 937,673 size 46x22; Text 'STOP'
   Button "Bouton_3" at 865,733 size 96x32; TextOff 'REST'
      on Press: SetBit("M_Reset")
      on Release: ResetBit("M_Reset")
   Switch "Commutateur_2" at 525,680 size 139x66; CaptionText 'Switch'; TextOff 'OFF'; TextOn 'ON'
      ProcessValue <- "M_Simulation"
      on SwitchOn: SetBit("M_Simulation")
      on SwitchOff: ResetBit("M_Simulation")
   SymbolLibrary "Bibliothèque des icônes_1" at 68,232 size 32x43
   SymbolLibrary "Bibliothèque des icônes_7" at 114,233 size 32x43
   Polyline "Ligne polygonale_3" at 394,190 size 56x50
      Visibility <- "Q_Xylanh_Do"
   Polyline "Ligne polygonale_4" at 394,184 size 61x51
      Visibility <- "Q_Xylanh_Do"
   Polyline "Ligne polygonale_1" at 755,195 size 56x50
      Visibility <- "Q_Xylanh_Xanh"
   Polyline "Ligne polygonale_2" at 755,189 size 61x51
      Visibility <- "Q_Xylanh_Xanh"
   Switch "Commutateur_3" at 0,364 size 108x52; CaptionText 'Switch'; TextOff 'OFF'; TextOn 'ON'
      on SwitchOn: SetBit("M_BT1")
      on SwitchOff: ResetBit("M_BT1")
      ProcessValue <- "M_BT1"
   Switch "Commutateur_4" at 828,361 size 108x52; TextOn 'ON'; CaptionText 'Switch'; TextOff 'OFF'
      on SwitchOff: ResetBit("M_BT2")
      on SwitchOn: SetBit("M_BT2")
      ProcessValue <- "M_BT2"
   Switch "Commutateur_5" at 504,150 size 76x56; TextOn 'ON'; CaptionText 'Switch'; TextOff 'OFF'
      on SwitchOff: ResetBit("M_Xylanh_Do")
      on SwitchOn: SetBit("M_Xylanh_Do")
      ProcessValue <- "M_Xylanh_Do"
   Switch "Commutateur_6" at 873,176 size 76x56; TextOn 'ON'; CaptionText 'Switch'; TextOff 'OFF'
      on SwitchOff: ResetBit("M_Xylanh_Xanh")
      on SwitchOn: SetBit("M_Xylanh_Xanh")
      ProcessValue <- "M_Xylanh_Xanh"
   Button "Bouton_4" at 284,474 size 96x32; TextOff 'Q PHAI'
      on Press: SetBit("M_Robot_Do_Phai")
      on Release: ResetBit("M_Robot_Do_Phai")
   Button "Bouton_5" at 293,512 size 96x32; TextOff 'GLUA'
      on Press: SetBit("M_Robot_Do_Glua")
      on Release: ResetBit("M_Robot_Do_Glua")
   Button "Bouton_6" at 302,550 size 96x32; TextOff 'Q TRAI'
      on Press: SetBit("M_Robot_Do_Trai")
      on Release: ResetBit("M_Robot_Do_Trai")
   Button "Bouton_7" at 657,470 size 96x32; TextOff 'Q PHAI'
      on Press: SetBit("M_Robot_Xanh_Phai")
      on Release: ResetBit("M_Robot_Xanh_Phai")
   Button "Bouton_8" at 666,508 size 96x32; TextOff 'GLUA'
      on Press: SetBit("M_Robot_Xanh_Glua")
      on Release: ResetBit("M_Robot_Xanh_Glua")
   Button "Bouton_9" at 675,546 size 96x32; TextOff 'Q TRAI'
      on Press: SetBit("M_Robot_Xanh_Trai")
      on Release: ResetBit("M_Robot_Xanh_Trai")
   Rectangle "Rectangle_17" at 480,335 size 51x19
      Visibility <- "Q_Robot_Xanh_Trai"
      Appearance <- "Q_Robot_Xanh_Trai"
   Polygon "Polygone_21" at 457,327 size 22x35
      Visibility <- "Q_Robot_Xanh_Trai"
      Appearance <- "Q_Robot_Xanh_Trai"
   Rectangle "Rectangle_18" at 595,343 size 51x19
      Appearance <- "Q_Robot_Xanh_Phai"
      Visibility <- "Q_Robot_Xanh_Phai"
   Polygon "Polygone_22" at 640,333 size 38x35
      Appearance <- "Q_Robot_Xanh_Phai"
      Visibility <- "Q_Robot_Xanh_Phai"
   Rectangle "Rectangle_19" at 124,325 size 51x19
      Visibility <- "Q_Robot_Do_Trai"
      Appearance <- "Q_Robot_Do_Trai"
   Polygon "Polygone_23" at 101,317 size 22x35
      Visibility <- "Q_Robot_Do_Trai"
      Appearance <- "Q_Robot_Do_Trai"
   Rectangle "Rectangle_20" at 239,333 size 51x19
      Appearance <- "Q_Robot_Do_Phai"
      Visibility <- "Q_Robot_Do_Phai"
   Polygon "Polygone_24" at 284,323 size 38x35
      Appearance <- "Q_Robot_Do_Phai"
      Visibility <- "Q_Robot_Do_Phai"
*)